FUNCTION_BLOCK BOOL_TO_QUARTER (* BOOL to quad-state *)
  (* Standard: 61499-2 *)
  (* Version 1.0, 2024-02-23, franz *)
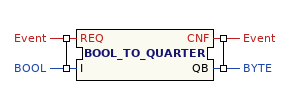
  EVENT_INPUT
    REQ WITH I; (* Normal Execution Request *)
  END_EVENT
  EVENT_OUTPUT
    CNF WITH QB; (* Execution Confirmation *)
  END_EVENT
  VAR_INPUT
    I : BOOL := FALSE; (* BOOL Input *)
  END_VAR
  VAR_OUTPUT
    QB : BYTE := COMMAND_DISABLE; (* 2bit (quarter Byte) Output with 4 States (only 2 used) *)
  END_VAR
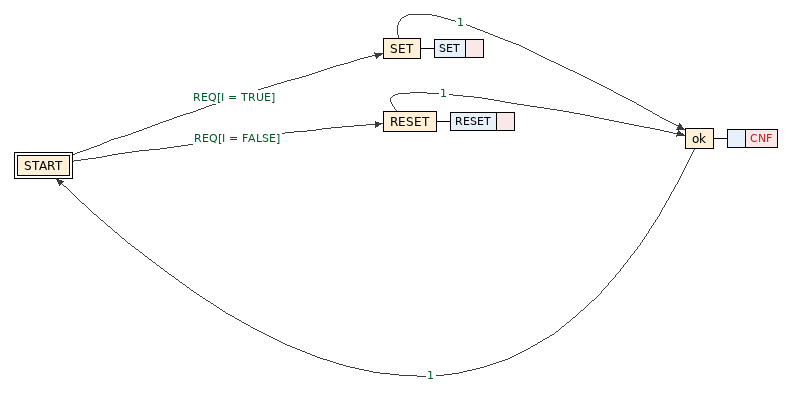
  EC_STATES
    START; (* Initial State *)
    SET : SET;
    RESET : RESET;
    ok : -> CNF;
  END_STATES
  EC_TRANSITIONS
    START TO SET := REQ[I = TRUE];
    START TO RESET := REQ[I = FALSE];
    SET TO ok := 1;
    RESET TO ok := 1;
    ok TO START := 1;
  END_TRANSITIONS
  ALGORITHM SET IN ST:
QB := COMMAND_ENABLE;
  END_ALGORITHM
  ALGORITHM RESET IN ST:
QB := COMMAND_DISABLE;
  END_ALGORITHM
END_FUNCTION_BLOCK
